# B&R Automation Studio project ABC_Pltzr (part 8)

#### S44paramCyclic.st
```iecst
(********************************************************************
 * COPYRIGHT --
 ********************************************************************
 * Program: S44param
 * File: S44paramCyclic.st
 * Author: scoccimaroj
 * Created: July 15, 2010
 ********************************************************************
 * Implementation of program S44param
 ********************************************************************)

PROGRAM _CYCLIC

CASE State OF

	(* Wait for a start command *)
	0:

		IF (cmdStart) THEN
			cmdStart :=	0;
			i := 0;
			State := 1;
		END_IF

	(* Reads the X64 parameter *)
	1:
		AsIOAccRead_0.enable :=	1;
		AsIOAccRead_0.pChannelName := ADR(S44ParRead.Parameters[i].ChannelName);

		(* If the status = 0, then the read was successful.  Store the value read. *)
		IF (AsIOAccRead_0.status = 0) THEN
			S44ParRead.Parameters[i].Data := AsIOAccRead_0.value;
			AsIOAccRead_0.enable :=	0;
			State := 2;

		(* Remain until the Read FUB is completed *)
		ELSIF (AsIOAccRead_0.status = ERR_FUB_BUSY) OR (AsIOAccRead_0.status = ERR_FUB_ENABLE_FALSE) THEN
			State := 1;

		(* If a FUB error occurs go to the next parameter *)
		ELSE
			AsIOAccRead_0.enable :=	0;
			State := 2;
		END_IF

	2:
		(* all the parameters have been read *)
		IF (i >= NUM_OF_S44PAR) THEN
  			i := 0;
			State := 3;

		(* read the next parameter in the list *)
		ELSE
			i := i + 1;
			State := 1;

		END_IF

	(* Do a csv search to allocate memory for the csv file. *)
	3:
		csvSearch.pStructName := csvInit.pStructName;
		csvSearch.NumOfStructs := csvInit.NumOfStructs;
		csvSearch.pStructMem := csvInit.pStructMem;
		csvSearch.MemLen := csvInit.MemCounter;
		csvSearch.FullNameLenght := 0;
		csvSearch.Separator := 44; (* ascii code for , *)
		csvSearch.Options := 0;
		csvSearch.FileHeader := HEADER;
		csvSearch.pMaschineNo := ADR('machine 1');
  		csvSearch.pComment := ADR('S44 parameter read file');
  		csvSearch.pVersion := ADR('v0.01');
  		csvSearch();

		(* successfully created the file for writing *)
		IF (csvSearch.status = 0) THEN
			State := 4;

		(* Error occured to abort the process *)
		ELSIF (csvSearch.status <> 0) AND (csvSearch.status <> 65535) THEN
			State := 0;

		END_IF

	(* Write the data to the csv file *)
	4:
		csvWrite.pFileName := ADR(S44ParRead.CsvFileName);
  		csvWrite.pDevice := ADR(S44ParRead.FileDevice);
  		csvWrite.pPath := ADR(S44ParRead.FilePath);
  		csvWrite.pStructMem := csvInit.pStructMem;
		csvWrite.MemLen := csvSearch.FileLen;
		csvWrite.Mode := FILE_OW;
		csvWrite();

		(* Write completed successfully *)
		IF (csvWrite.status = 0) THEN
  			State := 0;

		ELSIF (csvWrite.status <> 0) AND (csvWrite.status <> 65535) THEN
			State := 0;

		END_IF

END_CASE

(* Function Block Calls *)
AsIOAccRead_0();

END_PROGRAM
```

Listed in the project but not available here: Logical/Libraries/sscanf2, Logical/paiComponents/bglib/bgXmlRpcParser.h, Logical/paiComponents/bglib/bgBitUtilities.h, Logical/paiComponents/bglib/bgBufMemAlloc.c, Logical/paiComponents/bglib/bgDataStructures.c, Logical/paiComponents/bglib/bgdebugV2.h, Logical/paiComponents/bglib/bgdebug.h, Logical/paiComponents/bglib/bgfsig.h, Logical/paiComponents/bglib/bgfsig.c, Logical/paiComponents/bglib/bgftpclient.h, Logical/paiComponents/bglib/bgftpclient.c, Logical/paiComponents/bglib/bgftpclient_lib.c, Logical/paiComponents/bglib/bgHttpAppWeb.h, Logical/paiComponents/bglib/bgHttpAppWeb.c, Logical/paiComponents/bglib/bgHttpAppXmlRpc.h, Logical/paiComponents/bglib/bgHttpAppXmlRpc.c, Logical/paiComponents/bglib/bgHttpProtocol.h, Logical/paiComponents/bglib/bgHttpProtocol.c, Logical/paiComponents/bglib/bglibversion.h, Logical/paiComponents/bglib/bglib-1.c, Logical/paiComponents/bglib/bglib.c, Logical/paiComponents/bglib/bgPVLogger2.c, Logical/paiComponents/bglib/bgPVLogger3.c, Logical/paiComponents/bglib/bgSecMD5Signature.h, Logical/paiComponents/bglib/bgSecMD5Signature.c, Logical/paiComponents/bglib/bgsscanf.c, Logical/paiComponents/bglib/bgstatemachine.h, Logical/paiComponents/bglib/bgstatemachine.c, Logical/paiComponents/bglib/bgstring.h, Logical/paiComponents/bglib/bgTcpSocketClientServer.h, Logical/paiComponents/bglib/bgTcpSocketClient.c, Logical/paiComponents/bglib/bgTimer.h, Logical/paiComponents/bglib/bgTimer1ms.c, Logical/paiComponents/bglib/bgXmlRpcParser.c, Logical/paiComponents/bglib/bgPVSerializeJSON.h, Logical/paiComponents/bglib/bgPVSerializeJSON.c, Logical/paiComponents/bglib/bgPVSerialize.h, Logical/paiComponents/bglib/bgTelnetSrvr-astcpV2.c, Logical/paiComponents/Libraries/bglibas/bglibas.typ, Logical/paiComponents/paiBnRVFD/paiBnRVFD.typ, Logical/paiComponents/paiBnRVFD/paiBnRVFDX64ParRW.typ, Logical/paiComponents/paiBnRVFD/paiVFDX64ParRW.var, Logical/paiComponents/paiBnRVFD/paiVFDX64/paiVFDX64ParRW.c, Logical/paiComponents/paiTelnet/paiTelnet.typ, Logical/paiComponents/paiTelnet/paiTelnet.var, Logical/paiComponents/paiTelnet/paiTelnet, Logical/paiComponents/paiTemplate/paiHMI/paiConfigSys.typ, Logical/paiComponents/paiTemplate/paiHMI/paiHMI.typ, Logical/paiComponents/paiTemplate/paiHMI/paiConfig.var, Logical/paiComponents/paiTemplate/paiHMI/paiHMI.var, Logical/paiComponents/paiHmi/paiHmiAlert.c, Logical/paiComponents/paiHmi/paiHmiDialog.c, Logical/paiComponents/paiHmi/paiHmiSystemDateTime.c, Logical/Globals/Global.typ, Logical/Globals/Global.var, Logical/Globals/Alarms.typ, Logical/Globals/Alarms.var, Logical/Globals/MachineIO.typ, Logical/Globals/MachineIO.var, Logical/Globals/ConfigApp.var, Logical/MachineControl/vfdControl/vfdControl.c, Logical/MachineControl/palProc/palleteProcessor.c, Logical/MachineControl/appHmi, Logical/MachineControl/appDraw/appDraw.c, Logical/MachineControl/appDraw/appDraw.var, Logical/MachineControl/simonly, Logical/MachineControl/machmode, Logical/MachineControl/infcvidle/Cyclic.ld, Logical/MachineControl/infcvidle/Init.ld, Logical/MachineControl/infcvidle/Exit.ld, Logical/MachineControl/infcvidle/Types.typ, Logical/MachineControl/infcvidle/Variables.var, Logical/MachineControl/caseturner, Logical/MachineControl/rowforming/Init.ld, Logical/MachineControl/blades, Logical/MachineControl/retainbar, Logical/MachineControl/squaring, Logical/MachineControl/elevator, Logical/MachineControl/elevmove, Logical/MachineControl/palletinfdis, Logical/MachineControl/diofilter, Logical/appConfigAndRecipes/appCfgRecDefault.h, Logical/appConfigAndRecipes/appConfigAndRecipes.var, Logical/appConfigAndRecipes/appCfgRec/appCfgRec.c, Logical/paiComponents/paiFileService/paiPVSerDesMgr.c, Logical/ParameterDownload/CSV_File/CSV_File.typ, Logical/ParameterDownload/CSV_File/CSV_File.var, Logical/ParameterDownload/CSV_File/CSV_File.fun, Logical/ParameterDownload/CSV_File/CSV_InitCheckFile.ab, Logical/ParameterDownload/CSV_File/CSV_Init.ab, Logical/ParameterDownload/CSV_File/SearchFileName.ab, Logical/ParameterDownload/CSV_File/CSV_ReadFile.ab, Logical/ParameterDownload/CSV_File/ExListFile.ab, Logical/ParameterDownload/CSV_File/CSV_WriteFile.ab, Logical/ParameterDownload/P74_Download/P74param/P74param.typ, Logical/ParameterDownload/P74_Download/P74param/P74param.var, Logical/ParameterDownload/P84_Download/P84param/P84paramCyclic.st, Logical/ParameterDownload/P84_Download/P84param/P84paramInit.st, Logical/ParameterDownload/P84_Download/P84param/P84param.var
